{attribute 'GeneratedUsingTerminal: EL2258-0000-0017'}
{attribute addProperty BoxType "EL2258-0000-0017"}
{attribute addProperty Id "StatusAT %I*Status_642C2ED16"}
{attribute addProperty CRC "1405132427"}
{attribute addProperty Size "6"}
TYPE MTO_Inputs_Channel_53C09E8B EXTENDS TcoIo.InputBase_8311D824 :
STRUCT
	{attribute addProperty Name "Status"}
	Status AT %I* : Status_642C2ED1;
END_STRUCT
END_TYPE

(* stored: Version 1.2.0.0, ProductVersion 3.1.4024.11
   DUT MTO_Inputs_Channel_53C09E8B: Id {5202c80c-8bd1-43ee-b34a-d78401b3578e} *)
